// TIA Portal V17 export
// export: Created 2025-03-05T08:03:01.4817043Z, ExportSetting WithDefaults, DisplayName Totally Integrated Automation Portal, DisplayVersion V17 Update 8, DisplayName TIA Portal Openness, DisplayVersion V17 Update 8, DisplayName TIA Portal Version Control Interface, DisplayVersion V17, DisplayName SINAMICS Startdrive Advanced, DisplayVersion V17 SP2, DisplayName SINAMICS Startdrive G110M, G120, G120C, G120D, G120P, G115D, DisplayVersion V17 SP2, DisplayName SINAMICS Startdrive G130, G150, S120, S150, SINAMICS MV, S210, DisplayVersion V17 SP2, DisplayName STEP 7 Professional, DisplayVersion V17 Update 8, DisplayName SINUMERIK ONE STEP 7 Toolbox, DisplayVersion V17 Update 12, DisplayName SINUMERIK 840D sl STEP 7 Toolbox, DisplayVersion V17 Update 12, DisplayName STEP 7 Safety, DisplayVersion V17 Update 6, DisplayName WinCC Advanced, DisplayVersion V17 Update 8
FUNCTION "FC21014_POWDER_FEEDER_PROFINET" : Void   // FC21014, LAD
TITLE = FC21014 POWDER FEEDER PROFINET
{ S7_Optimized_Access := 'TRUE' }
VERSION : 0.1
// stored: AutoNumber false, IsIECCheckEnabled false, SetENOAutomatically false, UDAEnableTagReadback false
BEGIN

REGION Network 1: /////_UNIT_01_/////
END_REGION

REGION Network 2: CALL FB21014 POWDER FEEDER 1 PROFINET UNIT 01
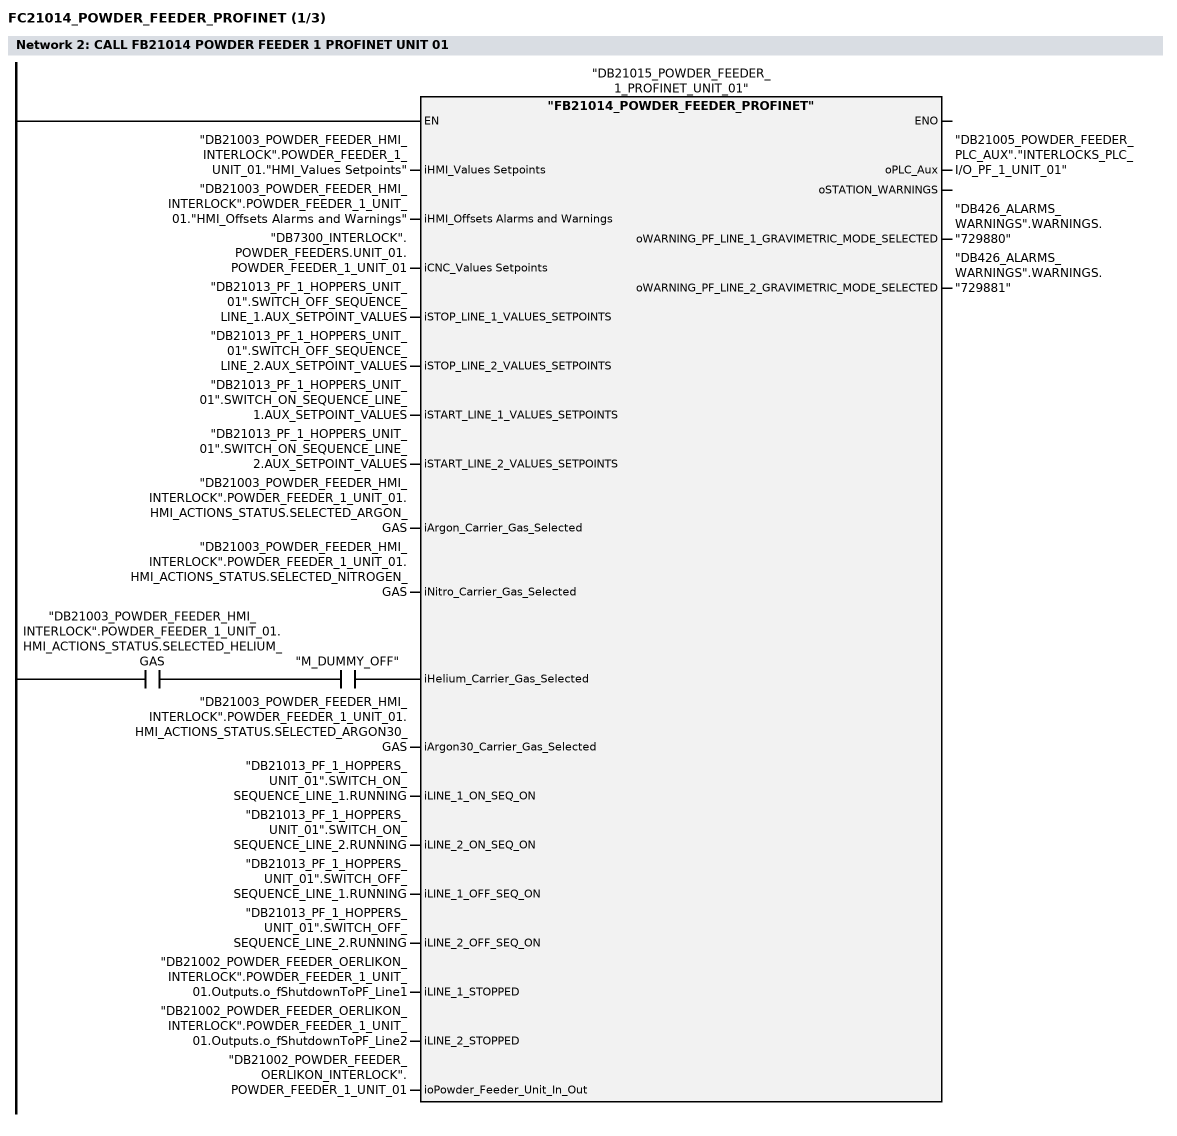
   RUNG wire#powerrail
      "DB21015_POWDER_FEEDER_1_PROFINET_UNIT_01"(iHelium_Carrier_Gas_Selected := wire#w1, "iHMI_Values Setpoints" := "DB21003_POWDER_FEEDER_HMI_INTERLOCK".POWDER_FEEDER_1_UNIT_01."HMI_Values Setpoints", "iHMI_Offsets Alarms and Warnings" := "DB21003_POWDER_FEEDER_HMI_INTERLOCK".POWDER_FEEDER_1_UNIT_01."HMI_Offsets Alarms and Warnings", "iCNC_Values Setpoints" := "DB7300_INTERLOCK".POWDER_FEEDERS.UNIT_01.POWDER_FEEDER_1_UNIT_01, iSTOP_LINE_1_VALUES_SETPOINTS := "DB21013_PF_1_HOPPERS_UNIT_01".SWITCH_OFF_SEQUENCE_LINE_1.AUX_SETPOINT_VALUES, iSTOP_LINE_2_VALUES_SETPOINTS := "DB21013_PF_1_HOPPERS_UNIT_01".SWITCH_OFF_SEQUENCE_LINE_2.AUX_SETPOINT_VALUES, iSTART_LINE_1_VALUES_SETPOINTS := "DB21013_PF_1_HOPPERS_UNIT_01".SWITCH_ON_SEQUENCE_LINE_1.AUX_SETPOINT_VALUES, iSTART_LINE_2_VALUES_SETPOINTS := "DB21013_PF_1_HOPPERS_UNIT_01".SWITCH_ON_SEQUENCE_LINE_2.AUX_SETPOINT_VALUES, iArgon_Carrier_Gas_Selected := "DB21003_POWDER_FEEDER_HMI_INTERLOCK".POWDER_FEEDER_1_UNIT_01.HMI_ACTIONS_STATUS.SELECTED_ARGON_GAS, iNitro_Carrier_Gas_Selected := "DB21003_POWDER_FEEDER_HMI_INTERLOCK".POWDER_FEEDER_1_UNIT_01.HMI_ACTIONS_STATUS.SELECTED_NITROGEN_GAS, iArgon30_Carrier_Gas_Selected := "DB21003_POWDER_FEEDER_HMI_INTERLOCK".POWDER_FEEDER_1_UNIT_01.HMI_ACTIONS_STATUS.SELECTED_ARGON30_GAS, iLINE_1_ON_SEQ_ON := "DB21013_PF_1_HOPPERS_UNIT_01".SWITCH_ON_SEQUENCE_LINE_1.RUNNING, iLINE_2_ON_SEQ_ON := "DB21013_PF_1_HOPPERS_UNIT_01".SWITCH_ON_SEQUENCE_LINE_2.RUNNING, iLINE_1_OFF_SEQ_ON := "DB21013_PF_1_HOPPERS_UNIT_01".SWITCH_OFF_SEQUENCE_LINE_1.RUNNING, iLINE_2_OFF_SEQ_ON := "DB21013_PF_1_HOPPERS_UNIT_01".SWITCH_OFF_SEQUENCE_LINE_2.RUNNING, iLINE_1_STOPPED := "DB21002_POWDER_FEEDER_OERLIKON_INTERLOCK".POWDER_FEEDER_1_UNIT_01.Outputs.o_fShutdownToPF_Line1, iLINE_2_STOPPED := "DB21002_POWDER_FEEDER_OERLIKON_INTERLOCK".POWDER_FEEDER_1_UNIT_01.Outputs.o_fShutdownToPF_Line2, ioPowder_Feeder_Unit_In_Out := "DB21002_POWDER_FEEDER_OERLIKON_INTERLOCK".POWDER_FEEDER_1_UNIT_01, oPLC_Aux => "DB21005_POWDER_FEEDER_PLC_AUX"."INTERLOCKS_PLC_I/O_PF_1_UNIT_01", oSTATION_WARNINGS =>, oWARNING_PF_LINE_1_GRAVIMETRIC_MODE_SELECTED => "DB426_ALARMS_WARNINGS".WARNINGS."729880", oWARNING_PF_LINE_2_GRAVIMETRIC_MODE_SELECTED => "DB426_ALARMS_WARNINGS".WARNINGS."729881")
   END_RUNG
   RUNG wire#powerrail
      Contact( "DB21003_POWDER_FEEDER_HMI_INTERLOCK".POWDER_FEEDER_1_UNIT_01.HMI_ACTIONS_STATUS.SELECTED_HELIUM_GAS )
      Contact( "M_DUMMY_OFF" )
   END_RUNG wire#w1
   // the same network as SCL:
   "DB21015_POWDER_FEEDER_1_PROFINET_UNIT_01"("iHMI_Values Setpoints" := "DB21003_POWDER_FEEDER_HMI_INTERLOCK".POWDER_FEEDER_1_UNIT_01."HMI_Values Setpoints",   // "FB21014_POWDER_FEEDER_PROFINET"
                           "iHMI_Offsets Alarms and Warnings" := "DB21003_POWDER_FEEDER_HMI_INTERLOCK".POWDER_FEEDER_1_UNIT_01."HMI_Offsets Alarms and Warnings",
                           "iCNC_Values Setpoints" := "DB7300_INTERLOCK".POWDER_FEEDERS.UNIT_01.POWDER_FEEDER_1_UNIT_01,
                           iSTOP_LINE_1_VALUES_SETPOINTS := "DB21013_PF_1_HOPPERS_UNIT_01".SWITCH_OFF_SEQUENCE_LINE_1.AUX_SETPOINT_VALUES,
                           iSTOP_LINE_2_VALUES_SETPOINTS := "DB21013_PF_1_HOPPERS_UNIT_01".SWITCH_OFF_SEQUENCE_LINE_2.AUX_SETPOINT_VALUES,
                           iSTART_LINE_1_VALUES_SETPOINTS := "DB21013_PF_1_HOPPERS_UNIT_01".SWITCH_ON_SEQUENCE_LINE_1.AUX_SETPOINT_VALUES,
                           iSTART_LINE_2_VALUES_SETPOINTS := "DB21013_PF_1_HOPPERS_UNIT_01".SWITCH_ON_SEQUENCE_LINE_2.AUX_SETPOINT_VALUES,
                           iArgon_Carrier_Gas_Selected := "DB21003_POWDER_FEEDER_HMI_INTERLOCK".POWDER_FEEDER_1_UNIT_01.HMI_ACTIONS_STATUS.SELECTED_ARGON_GAS,
                           iNitro_Carrier_Gas_Selected := "DB21003_POWDER_FEEDER_HMI_INTERLOCK".POWDER_FEEDER_1_UNIT_01.HMI_ACTIONS_STATUS.SELECTED_NITROGEN_GAS,
                           iHelium_Carrier_Gas_Selected := "DB21003_POWDER_FEEDER_HMI_INTERLOCK".POWDER_FEEDER_1_UNIT_01.HMI_ACTIONS_STATUS.SELECTED_HELIUM_GAS AND "M_DUMMY_OFF",
                           iArgon30_Carrier_Gas_Selected := "DB21003_POWDER_FEEDER_HMI_INTERLOCK".POWDER_FEEDER_1_UNIT_01.HMI_ACTIONS_STATUS.SELECTED_ARGON30_GAS,
                           iLINE_1_ON_SEQ_ON := "DB21013_PF_1_HOPPERS_UNIT_01".SWITCH_ON_SEQUENCE_LINE_1.RUNNING,
                           iLINE_2_ON_SEQ_ON := "DB21013_PF_1_HOPPERS_UNIT_01".SWITCH_ON_SEQUENCE_LINE_2.RUNNING,
                           iLINE_1_OFF_SEQ_ON := "DB21013_PF_1_HOPPERS_UNIT_01".SWITCH_OFF_SEQUENCE_LINE_1.RUNNING,
                           iLINE_2_OFF_SEQ_ON := "DB21013_PF_1_HOPPERS_UNIT_01".SWITCH_OFF_SEQUENCE_LINE_2.RUNNING,
                           iLINE_1_STOPPED := "DB21002_POWDER_FEEDER_OERLIKON_INTERLOCK".POWDER_FEEDER_1_UNIT_01.Outputs.o_fShutdownToPF_Line1,
                           iLINE_2_STOPPED := "DB21002_POWDER_FEEDER_OERLIKON_INTERLOCK".POWDER_FEEDER_1_UNIT_01.Outputs.o_fShutdownToPF_Line2,
                           ioPowder_Feeder_Unit_In_Out := "DB21002_POWDER_FEEDER_OERLIKON_INTERLOCK".POWDER_FEEDER_1_UNIT_01,
                           oPLC_Aux => "DB21005_POWDER_FEEDER_PLC_AUX"."INTERLOCKS_PLC_I/O_PF_1_UNIT_01",
                           oWARNING_PF_LINE_1_GRAVIMETRIC_MODE_SELECTED => "DB426_ALARMS_WARNINGS".WARNINGS."729880",
                           oWARNING_PF_LINE_2_GRAVIMETRIC_MODE_SELECTED => "DB426_ALARMS_WARNINGS".WARNINGS."729881");
END_REGION

REGION Network 3: /////_UNIT_02_/////
END_REGION

REGION Network 4: CALL FB21014 POWDER FEEDER 1 PROFINET UNIT 02
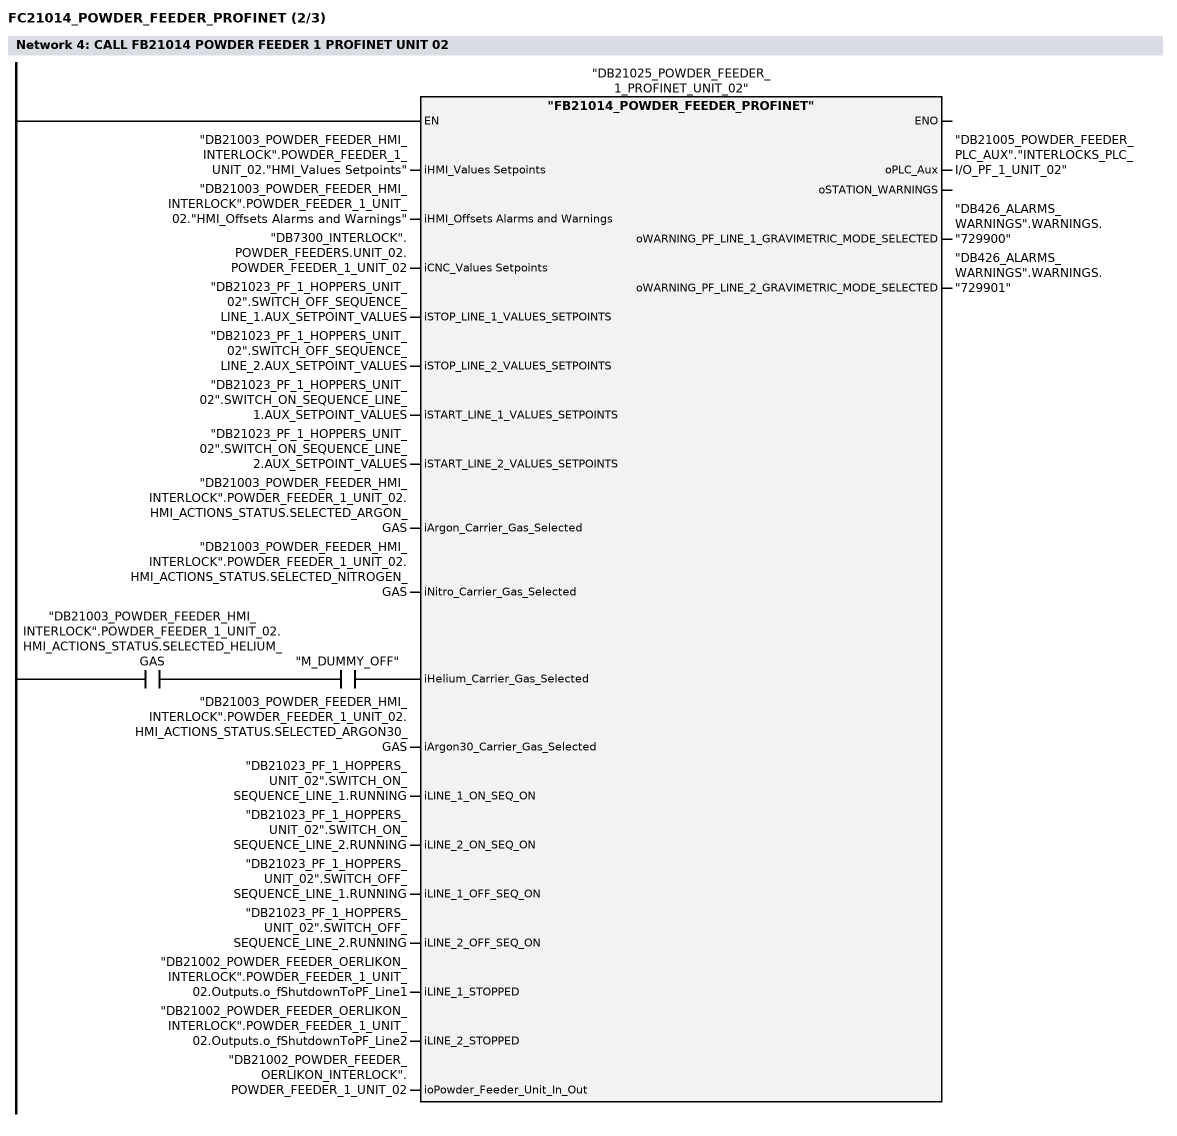
   RUNG wire#powerrail
      "DB21025_POWDER_FEEDER_1_PROFINET_UNIT_02"(iHelium_Carrier_Gas_Selected := wire#w1, "iHMI_Values Setpoints" := "DB21003_POWDER_FEEDER_HMI_INTERLOCK".POWDER_FEEDER_1_UNIT_02."HMI_Values Setpoints", "iHMI_Offsets Alarms and Warnings" := "DB21003_POWDER_FEEDER_HMI_INTERLOCK".POWDER_FEEDER_1_UNIT_02."HMI_Offsets Alarms and Warnings", "iCNC_Values Setpoints" := "DB7300_INTERLOCK".POWDER_FEEDERS.UNIT_02.POWDER_FEEDER_1_UNIT_02, iSTOP_LINE_1_VALUES_SETPOINTS := "DB21023_PF_1_HOPPERS_UNIT_02".SWITCH_OFF_SEQUENCE_LINE_1.AUX_SETPOINT_VALUES, iSTOP_LINE_2_VALUES_SETPOINTS := "DB21023_PF_1_HOPPERS_UNIT_02".SWITCH_OFF_SEQUENCE_LINE_2.AUX_SETPOINT_VALUES, iSTART_LINE_1_VALUES_SETPOINTS := "DB21023_PF_1_HOPPERS_UNIT_02".SWITCH_ON_SEQUENCE_LINE_1.AUX_SETPOINT_VALUES, iSTART_LINE_2_VALUES_SETPOINTS := "DB21023_PF_1_HOPPERS_UNIT_02".SWITCH_ON_SEQUENCE_LINE_2.AUX_SETPOINT_VALUES, iArgon_Carrier_Gas_Selected := "DB21003_POWDER_FEEDER_HMI_INTERLOCK".POWDER_FEEDER_1_UNIT_02.HMI_ACTIONS_STATUS.SELECTED_ARGON_GAS, iNitro_Carrier_Gas_Selected := "DB21003_POWDER_FEEDER_HMI_INTERLOCK".POWDER_FEEDER_1_UNIT_02.HMI_ACTIONS_STATUS.SELECTED_NITROGEN_GAS, iArgon30_Carrier_Gas_Selected := "DB21003_POWDER_FEEDER_HMI_INTERLOCK".POWDER_FEEDER_1_UNIT_02.HMI_ACTIONS_STATUS.SELECTED_ARGON30_GAS, iLINE_1_ON_SEQ_ON := "DB21023_PF_1_HOPPERS_UNIT_02".SWITCH_ON_SEQUENCE_LINE_1.RUNNING, iLINE_2_ON_SEQ_ON := "DB21023_PF_1_HOPPERS_UNIT_02".SWITCH_ON_SEQUENCE_LINE_2.RUNNING, iLINE_1_OFF_SEQ_ON := "DB21023_PF_1_HOPPERS_UNIT_02".SWITCH_OFF_SEQUENCE_LINE_1.RUNNING, iLINE_2_OFF_SEQ_ON := "DB21023_PF_1_HOPPERS_UNIT_02".SWITCH_OFF_SEQUENCE_LINE_2.RUNNING, iLINE_1_STOPPED := "DB21002_POWDER_FEEDER_OERLIKON_INTERLOCK".POWDER_FEEDER_1_UNIT_02.Outputs.o_fShutdownToPF_Line1, iLINE_2_STOPPED := "DB21002_POWDER_FEEDER_OERLIKON_INTERLOCK".POWDER_FEEDER_1_UNIT_02.Outputs.o_fShutdownToPF_Line2, ioPowder_Feeder_Unit_In_Out := "DB21002_POWDER_FEEDER_OERLIKON_INTERLOCK".POWDER_FEEDER_1_UNIT_02, oPLC_Aux => "DB21005_POWDER_FEEDER_PLC_AUX"."INTERLOCKS_PLC_I/O_PF_1_UNIT_02", oSTATION_WARNINGS =>, oWARNING_PF_LINE_1_GRAVIMETRIC_MODE_SELECTED => "DB426_ALARMS_WARNINGS".WARNINGS."729900", oWARNING_PF_LINE_2_GRAVIMETRIC_MODE_SELECTED => "DB426_ALARMS_WARNINGS".WARNINGS."729901")
   END_RUNG
   RUNG wire#powerrail
      Contact( "DB21003_POWDER_FEEDER_HMI_INTERLOCK".POWDER_FEEDER_1_UNIT_02.HMI_ACTIONS_STATUS.SELECTED_HELIUM_GAS )
      Contact( "M_DUMMY_OFF" )
   END_RUNG wire#w1
   // the same network as SCL:
   "DB21025_POWDER_FEEDER_1_PROFINET_UNIT_02"("iHMI_Values Setpoints" := "DB21003_POWDER_FEEDER_HMI_INTERLOCK".POWDER_FEEDER_1_UNIT_02."HMI_Values Setpoints",   // "FB21014_POWDER_FEEDER_PROFINET"
                           "iHMI_Offsets Alarms and Warnings" := "DB21003_POWDER_FEEDER_HMI_INTERLOCK".POWDER_FEEDER_1_UNIT_02."HMI_Offsets Alarms and Warnings",
                           "iCNC_Values Setpoints" := "DB7300_INTERLOCK".POWDER_FEEDERS.UNIT_02.POWDER_FEEDER_1_UNIT_02,
                           iSTOP_LINE_1_VALUES_SETPOINTS := "DB21023_PF_1_HOPPERS_UNIT_02".SWITCH_OFF_SEQUENCE_LINE_1.AUX_SETPOINT_VALUES,
                           iSTOP_LINE_2_VALUES_SETPOINTS := "DB21023_PF_1_HOPPERS_UNIT_02".SWITCH_OFF_SEQUENCE_LINE_2.AUX_SETPOINT_VALUES,
                           iSTART_LINE_1_VALUES_SETPOINTS := "DB21023_PF_1_HOPPERS_UNIT_02".SWITCH_ON_SEQUENCE_LINE_1.AUX_SETPOINT_VALUES,
                           iSTART_LINE_2_VALUES_SETPOINTS := "DB21023_PF_1_HOPPERS_UNIT_02".SWITCH_ON_SEQUENCE_LINE_2.AUX_SETPOINT_VALUES,
                           iArgon_Carrier_Gas_Selected := "DB21003_POWDER_FEEDER_HMI_INTERLOCK".POWDER_FEEDER_1_UNIT_02.HMI_ACTIONS_STATUS.SELECTED_ARGON_GAS,
                           iNitro_Carrier_Gas_Selected := "DB21003_POWDER_FEEDER_HMI_INTERLOCK".POWDER_FEEDER_1_UNIT_02.HMI_ACTIONS_STATUS.SELECTED_NITROGEN_GAS,
                           iHelium_Carrier_Gas_Selected := "DB21003_POWDER_FEEDER_HMI_INTERLOCK".POWDER_FEEDER_1_UNIT_02.HMI_ACTIONS_STATUS.SELECTED_HELIUM_GAS AND "M_DUMMY_OFF",
                           iArgon30_Carrier_Gas_Selected := "DB21003_POWDER_FEEDER_HMI_INTERLOCK".POWDER_FEEDER_1_UNIT_02.HMI_ACTIONS_STATUS.SELECTED_ARGON30_GAS,
                           iLINE_1_ON_SEQ_ON := "DB21023_PF_1_HOPPERS_UNIT_02".SWITCH_ON_SEQUENCE_LINE_1.RUNNING,
                           iLINE_2_ON_SEQ_ON := "DB21023_PF_1_HOPPERS_UNIT_02".SWITCH_ON_SEQUENCE_LINE_2.RUNNING,
                           iLINE_1_OFF_SEQ_ON := "DB21023_PF_1_HOPPERS_UNIT_02".SWITCH_OFF_SEQUENCE_LINE_1.RUNNING,
                           iLINE_2_OFF_SEQ_ON := "DB21023_PF_1_HOPPERS_UNIT_02".SWITCH_OFF_SEQUENCE_LINE_2.RUNNING,
                           iLINE_1_STOPPED := "DB21002_POWDER_FEEDER_OERLIKON_INTERLOCK".POWDER_FEEDER_1_UNIT_02.Outputs.o_fShutdownToPF_Line1,
                           iLINE_2_STOPPED := "DB21002_POWDER_FEEDER_OERLIKON_INTERLOCK".POWDER_FEEDER_1_UNIT_02.Outputs.o_fShutdownToPF_Line2,
                           ioPowder_Feeder_Unit_In_Out := "DB21002_POWDER_FEEDER_OERLIKON_INTERLOCK".POWDER_FEEDER_1_UNIT_02,
                           oPLC_Aux => "DB21005_POWDER_FEEDER_PLC_AUX"."INTERLOCKS_PLC_I/O_PF_1_UNIT_02",
                           oWARNING_PF_LINE_1_GRAVIMETRIC_MODE_SELECTED => "DB426_ALARMS_WARNINGS".WARNINGS."729900",
                           oWARNING_PF_LINE_2_GRAVIMETRIC_MODE_SELECTED => "DB426_ALARMS_WARNINGS".WARNINGS."729901");
END_REGION

REGION Network 5: CALL FB21014 POWDER FEEDER 2 PROFINET UNIT 02
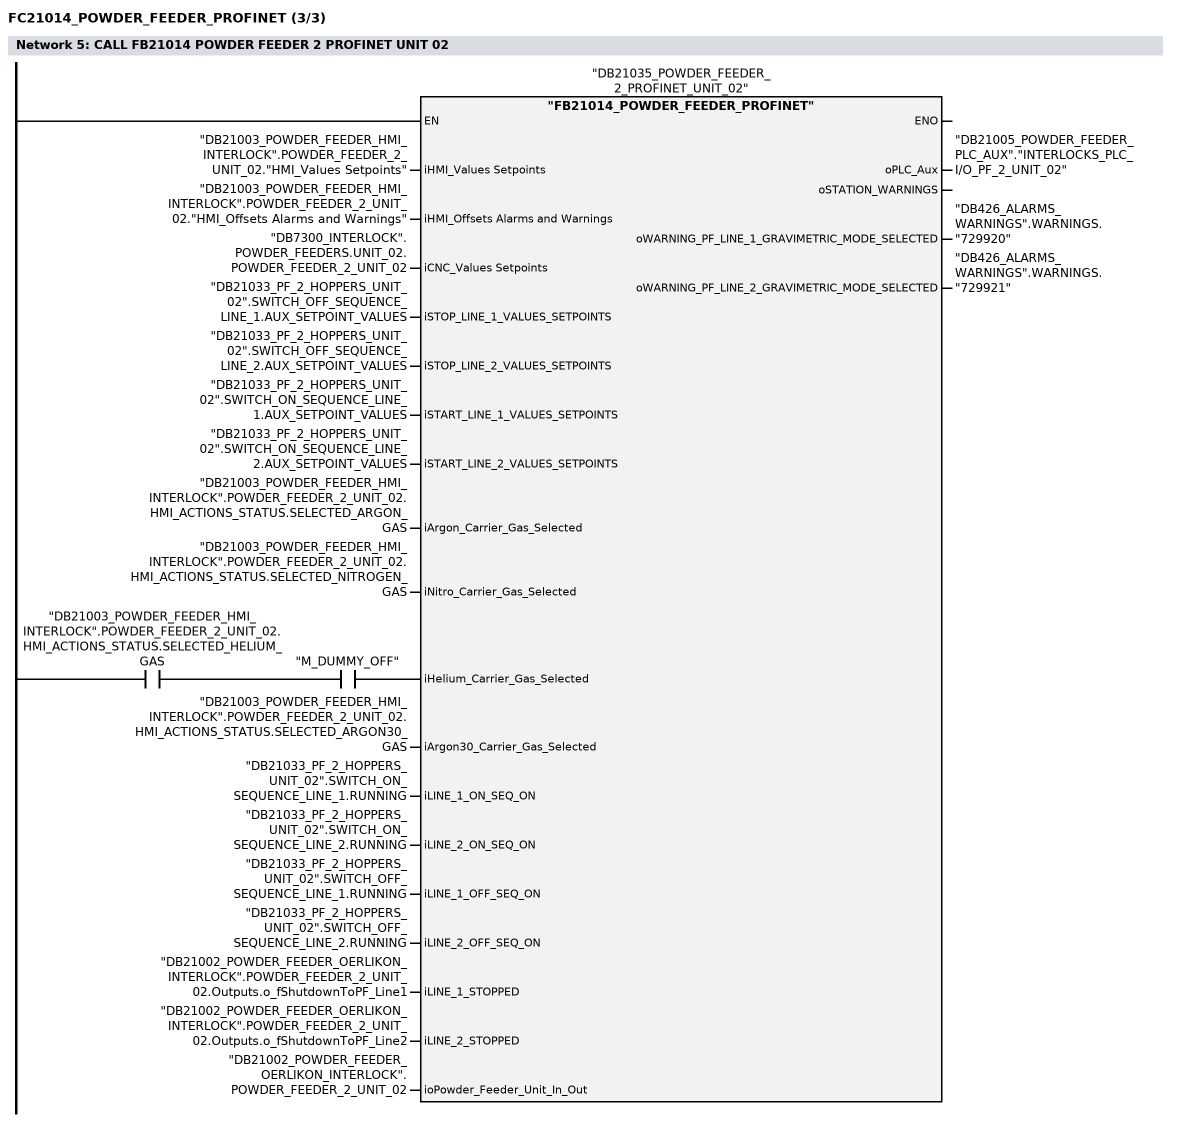
   RUNG wire#powerrail
      "DB21035_POWDER_FEEDER_2_PROFINET_UNIT_02"(iHelium_Carrier_Gas_Selected := wire#w1, "iHMI_Values Setpoints" := "DB21003_POWDER_FEEDER_HMI_INTERLOCK".POWDER_FEEDER_2_UNIT_02."HMI_Values Setpoints", "iHMI_Offsets Alarms and Warnings" := "DB21003_POWDER_FEEDER_HMI_INTERLOCK".POWDER_FEEDER_2_UNIT_02."HMI_Offsets Alarms and Warnings", "iCNC_Values Setpoints" := "DB7300_INTERLOCK".POWDER_FEEDERS.UNIT_02.POWDER_FEEDER_2_UNIT_02, iSTOP_LINE_1_VALUES_SETPOINTS := "DB21033_PF_2_HOPPERS_UNIT_02".SWITCH_OFF_SEQUENCE_LINE_1.AUX_SETPOINT_VALUES, iSTOP_LINE_2_VALUES_SETPOINTS := "DB21033_PF_2_HOPPERS_UNIT_02".SWITCH_OFF_SEQUENCE_LINE_2.AUX_SETPOINT_VALUES, iSTART_LINE_1_VALUES_SETPOINTS := "DB21033_PF_2_HOPPERS_UNIT_02".SWITCH_ON_SEQUENCE_LINE_1.AUX_SETPOINT_VALUES, iSTART_LINE_2_VALUES_SETPOINTS := "DB21033_PF_2_HOPPERS_UNIT_02".SWITCH_ON_SEQUENCE_LINE_2.AUX_SETPOINT_VALUES, iArgon_Carrier_Gas_Selected := "DB21003_POWDER_FEEDER_HMI_INTERLOCK".POWDER_FEEDER_2_UNIT_02.HMI_ACTIONS_STATUS.SELECTED_ARGON_GAS, iNitro_Carrier_Gas_Selected := "DB21003_POWDER_FEEDER_HMI_INTERLOCK".POWDER_FEEDER_2_UNIT_02.HMI_ACTIONS_STATUS.SELECTED_NITROGEN_GAS, iArgon30_Carrier_Gas_Selected := "DB21003_POWDER_FEEDER_HMI_INTERLOCK".POWDER_FEEDER_2_UNIT_02.HMI_ACTIONS_STATUS.SELECTED_ARGON30_GAS, iLINE_1_ON_SEQ_ON := "DB21033_PF_2_HOPPERS_UNIT_02".SWITCH_ON_SEQUENCE_LINE_1.RUNNING, iLINE_2_ON_SEQ_ON := "DB21033_PF_2_HOPPERS_UNIT_02".SWITCH_ON_SEQUENCE_LINE_2.RUNNING, iLINE_1_OFF_SEQ_ON := "DB21033_PF_2_HOPPERS_UNIT_02".SWITCH_OFF_SEQUENCE_LINE_1.RUNNING, iLINE_2_OFF_SEQ_ON := "DB21033_PF_2_HOPPERS_UNIT_02".SWITCH_OFF_SEQUENCE_LINE_2.RUNNING, iLINE_1_STOPPED := "DB21002_POWDER_FEEDER_OERLIKON_INTERLOCK".POWDER_FEEDER_2_UNIT_02.Outputs.o_fShutdownToPF_Line1, iLINE_2_STOPPED := "DB21002_POWDER_FEEDER_OERLIKON_INTERLOCK".POWDER_FEEDER_2_UNIT_02.Outputs.o_fShutdownToPF_Line2, ioPowder_Feeder_Unit_In_Out := "DB21002_POWDER_FEEDER_OERLIKON_INTERLOCK".POWDER_FEEDER_2_UNIT_02, oPLC_Aux => "DB21005_POWDER_FEEDER_PLC_AUX"."INTERLOCKS_PLC_I/O_PF_2_UNIT_02", oSTATION_WARNINGS =>, oWARNING_PF_LINE_1_GRAVIMETRIC_MODE_SELECTED => "DB426_ALARMS_WARNINGS".WARNINGS."729920", oWARNING_PF_LINE_2_GRAVIMETRIC_MODE_SELECTED => "DB426_ALARMS_WARNINGS".WARNINGS."729921")
   END_RUNG
   RUNG wire#powerrail
      Contact( "DB21003_POWDER_FEEDER_HMI_INTERLOCK".POWDER_FEEDER_2_UNIT_02.HMI_ACTIONS_STATUS.SELECTED_HELIUM_GAS )
      Contact( "M_DUMMY_OFF" )
   END_RUNG wire#w1
   // the same network as SCL:
   "DB21035_POWDER_FEEDER_2_PROFINET_UNIT_02"("iHMI_Values Setpoints" := "DB21003_POWDER_FEEDER_HMI_INTERLOCK".POWDER_FEEDER_2_UNIT_02."HMI_Values Setpoints",   // "FB21014_POWDER_FEEDER_PROFINET"
                           "iHMI_Offsets Alarms and Warnings" := "DB21003_POWDER_FEEDER_HMI_INTERLOCK".POWDER_FEEDER_2_UNIT_02."HMI_Offsets Alarms and Warnings",
                           "iCNC_Values Setpoints" := "DB7300_INTERLOCK".POWDER_FEEDERS.UNIT_02.POWDER_FEEDER_2_UNIT_02,
                           iSTOP_LINE_1_VALUES_SETPOINTS := "DB21033_PF_2_HOPPERS_UNIT_02".SWITCH_OFF_SEQUENCE_LINE_1.AUX_SETPOINT_VALUES,
                           iSTOP_LINE_2_VALUES_SETPOINTS := "DB21033_PF_2_HOPPERS_UNIT_02".SWITCH_OFF_SEQUENCE_LINE_2.AUX_SETPOINT_VALUES,
                           iSTART_LINE_1_VALUES_SETPOINTS := "DB21033_PF_2_HOPPERS_UNIT_02".SWITCH_ON_SEQUENCE_LINE_1.AUX_SETPOINT_VALUES,
                           iSTART_LINE_2_VALUES_SETPOINTS := "DB21033_PF_2_HOPPERS_UNIT_02".SWITCH_ON_SEQUENCE_LINE_2.AUX_SETPOINT_VALUES,
                           iArgon_Carrier_Gas_Selected := "DB21003_POWDER_FEEDER_HMI_INTERLOCK".POWDER_FEEDER_2_UNIT_02.HMI_ACTIONS_STATUS.SELECTED_ARGON_GAS,
                           iNitro_Carrier_Gas_Selected := "DB21003_POWDER_FEEDER_HMI_INTERLOCK".POWDER_FEEDER_2_UNIT_02.HMI_ACTIONS_STATUS.SELECTED_NITROGEN_GAS,
                           iHelium_Carrier_Gas_Selected := "DB21003_POWDER_FEEDER_HMI_INTERLOCK".POWDER_FEEDER_2_UNIT_02.HMI_ACTIONS_STATUS.SELECTED_HELIUM_GAS AND "M_DUMMY_OFF",
                           iArgon30_Carrier_Gas_Selected := "DB21003_POWDER_FEEDER_HMI_INTERLOCK".POWDER_FEEDER_2_UNIT_02.HMI_ACTIONS_STATUS.SELECTED_ARGON30_GAS,
                           iLINE_1_ON_SEQ_ON := "DB21033_PF_2_HOPPERS_UNIT_02".SWITCH_ON_SEQUENCE_LINE_1.RUNNING,
                           iLINE_2_ON_SEQ_ON := "DB21033_PF_2_HOPPERS_UNIT_02".SWITCH_ON_SEQUENCE_LINE_2.RUNNING,
                           iLINE_1_OFF_SEQ_ON := "DB21033_PF_2_HOPPERS_UNIT_02".SWITCH_OFF_SEQUENCE_LINE_1.RUNNING,
                           iLINE_2_OFF_SEQ_ON := "DB21033_PF_2_HOPPERS_UNIT_02".SWITCH_OFF_SEQUENCE_LINE_2.RUNNING,
                           iLINE_1_STOPPED := "DB21002_POWDER_FEEDER_OERLIKON_INTERLOCK".POWDER_FEEDER_2_UNIT_02.Outputs.o_fShutdownToPF_Line1,
                           iLINE_2_STOPPED := "DB21002_POWDER_FEEDER_OERLIKON_INTERLOCK".POWDER_FEEDER_2_UNIT_02.Outputs.o_fShutdownToPF_Line2,
                           ioPowder_Feeder_Unit_In_Out := "DB21002_POWDER_FEEDER_OERLIKON_INTERLOCK".POWDER_FEEDER_2_UNIT_02,
                           oPLC_Aux => "DB21005_POWDER_FEEDER_PLC_AUX"."INTERLOCKS_PLC_I/O_PF_2_UNIT_02",
                           oWARNING_PF_LINE_1_GRAVIMETRIC_MODE_SELECTED => "DB426_ALARMS_WARNINGS".WARNINGS."729920",
                           oWARNING_PF_LINE_2_GRAVIMETRIC_MODE_SELECTED => "DB426_ALARMS_WARNINGS".WARNINGS."729921");
END_REGION
END_FUNCTION
